TYPE NETWORK_BUFFER_SHORT :
STRUCT
	SIZE : UINT;
	BUFFER : NW_BUF_SHORT;
END_STRUCT
END_TYPE

(* stored: Version 1.1.0.1, ProductVersion 3.1.4022.7
   DUT NETWORK_BUFFER_SHORT: Id {6e1bc9ed-8231-480a-be80-394a9e766d9c} *)
